// TIA Portal V17 export
// export: Created 2025-06-26T07:49:55.5315592Z, ExportSetting WithDefaults, DisplayName Totally Integrated Automation Portal, DisplayVersion V17 Update 8, DisplayName TIA Portal Openness, DisplayVersion V17 Update 8, DisplayName TIA Portal Version Control Interface, DisplayVersion V17, DisplayName STEP 7 Professional, DisplayVersion V17 Update 8, DisplayName STEP 7 Safety, DisplayVersion V17 Update 6, DisplayName WinCC Advanced, DisplayVersion V17 Update 8
TYPE "stPerformanceControl"
// stored: IsFailsafeCompliant false
   STRUCT
      RunningCondition : Bool;   // 1 = motor run, 0 = motor stop
      RestrictionID : Int;   // Currently active restriction
      TargetValue : Real;   // Currently selected setpoint [C]
      CurrentValue : Real;   // Currently selected process value [C]
      fOut : Real;   // Compressor performance setpoint [%]
      Settings : "PerformanceControl-STRUCT";
      ManualMode : Struct
         ForceMaxPower : Bool;
         ForceMaxPowerAll : Bool;
         ForcePowerSetpoint : Bool;
         ForcePowerSetpointValue : Real;
      END_STRUCT;
   END_STRUCT;
   // // Settings.SwitchToStandby_timeDelay : Time until MinimumPerformnceRate leads to standby
END_TYPE
